FUNCTION_BLOCK FINAL PWMDemandedSpeedCalculator IMPLEMENTS DemandedSpeedInterface
VAR
	iInputSpeedBits AT %I* : ARRAY [1..BitArraySize] OF BYTE;
END_VAR
VAR CONSTANT
	// Array Length
	BitArraySize : UINT := 125;
	// PWM frequency
	PWMFrequency : UINT := 200;
    // PWM period
	PWMPeriod : REAL := 1 / PWMFrequency;
	// Microseconds in Frequency
	UsInFrequency : UDINT :=  Constants.OneSecondInUs / PWMFrequency;	
END_VAR

METHOD GetSpeed : UINT
VAR_INST
	TempSpindleSpeed : UINT;
	LastDemandedSpeed : UINT;
	TotalOnTime : UDINT;
	TotalOffTime : UDINT;
	DutyCycle : LREAL;
	DutyCycles : ARRAY [0..20] OF LREAL;
	MovingAverage : FB_MovingAverageReal;
	Scaling : FB_ScaleBetween;
END_VAR
VAR
	I : UINT;	
	J: UINT;
	BitMask : UINT;
	MaskedBit : BOOL;
END_VAR
// The input here is a PWM signal with a frequency of 200, a low of 1% duty, and a high of 95% duty.
// Basic Calculation for PWM pulses

 FOR I := 1 TO BitArraySize BY 1 DO
	 FOR J := 0 TO 7 BY 1 DO
		BitMask := SHL(1, J);
		MaskedBit := TO_BOOL(iInputSpeedBits[I] AND BitMask);
		IF MaskedBit THEN
			TotalOnTime := TotalOnTime + 1;
		ELSE
			TotalOffTime := TotalOffTime + 1; 
		END_IF
		// Stop at the end of the period
		IF (TotalOnTime + TotalOffTime) > UsInFrequency THEN
			EXIT;
		END_IF 
	 END_FOR
 END_FOR
 
// See if the period is up
IF (TotalOnTime + TotalOffTime) > UsInFrequency  THEN
	DutyCycle := TO_LREAL(TotalOnTime) / TO_LREAL(TotalOnTime + TotalOffTime);
	TotalOnTime := 0;
	TotalOffTime := 0;
	// Average the duty cycle and then scale the average
	MovingAverage(ValueToAdd := DutyCycle, 
				  AverageArray := DutyCycles);
	Scaling(RawValue:=MovingAverage.CurrentValue, RawValueMin:=0.0, 
					  RawValueMax:=1, ScaledValueMin:=0,
					  ScaledValueMax:=24000);
	LastDemandedSpeed := TO_UINT(Scaling.ScaledValue);
END_IF
GetSpeed := LastDemandedSpeed;
END_METHOD

END_FUNCTION_BLOCK

(* stored: Version 1.1.0.1, ProductVersion 3.1.4022.16
   POU PWMDemandedSpeedCalculator: Id {d7b7f4ec-2f11-4936-85ca-0e73dfdbc7ef}, SpecialFunc None
   Method GetSpeed: Id {213d3359-88cd-493d-995f-9cc6a93b1330} *)
